(* IEC 61131-3 sources: trust-platform/crates/trust-runtime/tests/fixtures/complete_program, 6 files *)

(* ---- types.st ---- *)
TYPE Color :
(
    Red := 0,
    Green := 1,
    Blue := 2
);
END_TYPE

NAMESPACE DemoTypes
TYPE Sensor :
STRUCT
    id : DINT;
    label : STRING[32];
    active : BOOL;
    value : REAL;
END_STRUCT
END_TYPE

TYPE ValueArray : ARRAY[0..3] OF DINT; END_TYPE
END_NAMESPACE

(* ---- api.st ---- *)
NAMESPACE DemoApi
INTERFACE IMotor
    METHOD Start : BOOL
    VAR_INPUT
        speed : DINT;
    END_VAR
    END_METHOD

    METHOD Stop : BOOL
    END_METHOD

    PROPERTY Speed : DINT
        GET
        END_GET
        SET
        END_SET
    END_PROPERTY
END_INTERFACE
END_NAMESPACE

(* ---- impl.st ---- *)
NAMESPACE DemoImpl

CLASS Motor IMPLEMENTS DemoApi.IMotor
VAR
    speed_value : DINT := 0;
    running : BOOL := FALSE;
END_VAR

METHOD PUBLIC Start : BOOL
VAR_INPUT
    speed : DINT;
END_VAR
speed_value := speed;
running := TRUE;
Start := running;
END_METHOD

METHOD PUBLIC Stop : BOOL
running := FALSE;
Stop := running;
END_METHOD

PUBLIC PROPERTY Speed : DINT
GET
    Speed := speed_value;
END_GET
SET
    speed_value := Speed;
END_SET
END_PROPERTY
END_CLASS
END_NAMESPACE

(* ---- lib.st ---- *)
NAMESPACE DemoLib
FUNCTION Add : DINT
VAR_INPUT
    A : DINT;
    B : DINT;
END_VAR
Add := A + B;
END_FUNCTION

FUNCTION SwapDint : BOOL
VAR_IN_OUT
    A : DINT;
    B : DINT;
END_VAR
VAR_TEMP
    temp : DINT;
END_VAR
temp := A;
A := B;
B := temp;
SwapDint := TRUE;
END_FUNCTION

FUNCTION_BLOCK FB_Accumulator
VAR_INPUT
    In : DINT;
END_VAR
VAR_OUTPUT
    Sum : DINT;
END_VAR
Sum := Sum + In;
END_FUNCTION_BLOCK
END_NAMESPACE

(* ---- config.st ---- *)
CONFIGURATION DemoConfig
VAR_GLOBAL
    gCounter : DINT := 0;
END_VAR
TASK Fast (INTERVAL := T#20ms, PRIORITY := 1);
PROGRAM Inst WITH Fast : MainProg;
END_CONFIGURATION

(* ---- main.st ---- *)
PROGRAM MainProg
VAR
    motor : DemoImpl.Motor;
    sensor : DemoTypes.Sensor;
    values : DemoTypes.ValueArray;
    acc : DemoLib.FB_Accumulator;
    sum : DINT := 0;
    total : DINT := 0;
    color : Color := Color#Red;
    swap_a : DINT := 10;
    swap_b : DINT := 20;
    ok : BOOL := FALSE;
END_VAR

ok := motor.Start(100);
motor.Speed := 100;
ok := motor.Stop();

sensor.id := 1;
sensor.label := 'Main';
sensor.active := TRUE;
sensor.value := REAL#12.5;

values[0] := DINT#1;
values[1] := DINT#2;
values[2] := DINT#3;
values[3] := DINT#4;

sum := DemoLib.Add(A := values[0], B := values[1]);
acc(In := sum);
total := acc.Sum;
ok := DemoLib.SwapDint(swap_a, swap_b);

IF ok THEN
    total := total + swap_a + swap_b;
    color := Color#Green;
END_IF;
END_PROGRAM
